INTERFACE I_Sensor

PROPERTY isActive : BOOL
GET
END_GET
END_PROPERTY

END_INTERFACE

(* stored: Version 1.1.0.1, ProductVersion 3.1.4024.12
   Itf I_Sensor: Id {3436fc6a-a421-440f-aa83-64d3c3069457}
   Property isActive: Id {cb758539-67dd-469e-ba0d-b450bb1df838}
   Get Get: Id {174d9b7c-ea0b-402e-a540-40310783ccd4} *)
